FUNCTION Convert_BOOL_TO_LWORD : BOOL
VAR_INPUT
	in : BOOL;
	out : REFERENCE TO LWORD;
END_VAR

out := BOOL_TO_LWORD(in);
Convert_BOOL_TO_LWORD := TRUE;

END_FUNCTION

(* stored: Version 1.1.0.1, ProductVersion 3.1.4024.12
   POU Convert_BOOL_TO_LWORD: Id {9cf55fc5-b6d1-4a16-a559-ac98c73a8663}, SpecialFunc None *)
